FUNCTION_BLOCK FB_ConfigPackage
VAR_INPUT
    bReloadDefaults : BOOL;
END_VAR
VAR_OUTPUT
    stMachineConfig : ST_MachineConfig;
    bSimulationMode : BOOL;
    bConfigValid : BOOL;
    bConfigChanged : BOOL;
    sValidationError : STRING(120);
END_VAR
VAR
    bInitialized : BOOL;
    rtrigReload : R_TRIG;
    nAxis : UINT;
END_VAR

rtrigReload(CLK := bReloadDefaults);
bConfigChanged := FALSE;

IF (NOT bInitialized) OR rtrigReload.Q THEN
    stMachineConfig.bSimulationMode := TRUE;
    stMachineConfig.nAxisCount := 2;

    FOR nAxis := 1 TO cMAX_AXES DO
        stMachineConfig.astAxisConfig[nAxis].fMaxVelocity := 500.0;
        stMachineConfig.astAxisConfig[nAxis].fMaxAcceleration := 2000.0;
        stMachineConfig.astAxisConfig[nAxis].fMaxDeceleration := 2000.0;
        stMachineConfig.astAxisConfig[nAxis].fJerkLimit := 10000.0;
        stMachineConfig.astAxisConfig[nAxis].fSoftLimitPositive := 300.0;
        stMachineConfig.astAxisConfig[nAxis].fSoftLimitNegative := -10.0;
        stMachineConfig.astAxisConfig[nAxis].fHomingVelocity := 50.0;
        stMachineConfig.astAxisConfig[nAxis].fHomingBackoffVelocity := 10.0;
        stMachineConfig.astAxisConfig[nAxis].bHomingDirectionPositive := FALSE;
        stMachineConfig.astAxisConfig[nAxis].fHomeOffset := 0.0;
        stMachineConfig.astAxisConfig[nAxis].fPositionErrorLimit := 2.0;
        stMachineConfig.astAxisConfig[nAxis].fJogVelocity := 100.0;
    END_FOR

    stMachineConfig.stSafetyConfig.tEStopDebounceTime := T#100MS;
    stMachineConfig.stSafetyConfig.tRelayDiscrepancyWindow := T#500MS;
    stMachineConfig.stSafetyConfig.tLimitDebounceTime := T#50MS;
    stMachineConfig.stSafetyConfig.tStuckSensorTimeout := T#5S;
    stMachineConfig.stTimingConfig.tInitTimeout := T#10S;
    stMachineConfig.stTimingConfig.tHomingTimeout := T#60S;
    stMachineConfig.stTimingConfig.tHomingStepTimeout := T#15S;
    stMachineConfig.stTimingConfig.nHomingMaxRetries := 2;
    stMachineConfig.stTimingConfig.tCommandTimeout := T#5S;
    stMachineConfig.stTimingConfig.tTestSettleTime := T#500MS;
    stMachineConfig.stTimingConfig.tTestStepTimeout := T#30S;
    stMachineConfig.stTraceConfig.nBufferSize := cTRACE_BUFFER_SIZE;
    stMachineConfig.stTraceConfig.nDisplayCount := cTRACE_DISPLAY_COUNT;
    stMachineConfig.stTraceConfig.nPendingQueueMax := cTRACE_PENDING_MAX;
    stMachineConfig.stAlarmConfig.nMaxActiveAlarms := cMAX_ALARMS;
    stMachineConfig.stAlarmConfig.nMaxAlarmHistory := cMAX_ALARM_HISTORY;

    bInitialized := TRUE;
    bConfigChanged := TRUE;
END_IF

bConfigValid := TRUE;
sValidationError := '';

IF (stMachineConfig.nAxisCount = 0) OR (stMachineConfig.nAxisCount > cMAX_AXES) THEN
    bConfigValid := FALSE;
    sValidationError := 'Axis count is outside supported range';
END_IF

(* Always use the compile-time array bound here. If a corrupt or externally
   loaded axis count exceeds cMAX_AXES, iterating to that value would access
   outside astAxisConfig before the invalid configuration could be rejected. *)
FOR nAxis := 1 TO cMAX_AXES DO
    IF nAxis <= stMachineConfig.nAxisCount THEN
        IF stMachineConfig.astAxisConfig[nAxis].fMaxVelocity <= 0.0 THEN
            bConfigValid := FALSE;
            sValidationError := 'Maximum velocity must be positive';
        ELSIF stMachineConfig.astAxisConfig[nAxis].fMaxAcceleration <= 0.0 THEN
            bConfigValid := FALSE;
            sValidationError := 'Maximum acceleration must be positive';
        ELSIF stMachineConfig.astAxisConfig[nAxis].fMaxDeceleration <= 0.0 THEN
            bConfigValid := FALSE;
            sValidationError := 'Maximum deceleration must be positive';
        ELSIF stMachineConfig.astAxisConfig[nAxis].fSoftLimitPositive <=
                stMachineConfig.astAxisConfig[nAxis].fSoftLimitNegative THEN
            bConfigValid := FALSE;
            sValidationError := 'Positive soft limit must exceed negative soft limit';
        END_IF
    END_IF
END_FOR

IF (stMachineConfig.stTimingConfig.tInitTimeout <= T#0MS) OR
   (stMachineConfig.stTimingConfig.tHomingTimeout <= T#0MS) OR
   (stMachineConfig.stTimingConfig.tCommandTimeout <= T#0MS) THEN
    bConfigValid := FALSE;
    sValidationError := 'Configured timeout must be greater than zero';
END_IF

bSimulationMode := stMachineConfig.bSimulationMode;

END_FUNCTION_BLOCK

(* stored: Version 1.1.0.1
   POU FB_ConfigPackage: Id {A5AEB081-B795-811A-3F02-6B8001AB0F88} *)
